(* IEC 61131-3 sources: AI4Industrial_Automation-FIRE2026/analysis/probe_reference, 30 files *)

(* ---- task_01.st ---- *)
PROGRAM T01
VAR_INPUT
    Low_Level_Sensor : BOOL;
    High_Level_Sensor : BOOL;
    Start_Button : BOOL;
    Stop_Button : BOOL;
END_VAR
VAR_OUTPUT
    Fill_Pump : BOOL;
END_VAR
Fill_Pump := ((Start_Button AND NOT Low_Level_Sensor) OR Fill_Pump) AND NOT High_Level_Sensor AND NOT Stop_Button;
END_PROGRAM

(* ---- task_02.st ---- *)
PROGRAM T02
VAR_OUTPUT
    Red_Light : BOOL;
    Yellow_Light : BOOL;
    Green_Light : BOOL;
END_VAR
VAR
    Cyc : TON;
    Restart : BOOL;
END_VAR
Cyc(IN := NOT Restart, PT := T#12s);
Restart := Cyc.Q;
Red_Light := Cyc.ET < T#5s;
Green_Light := Cyc.ET >= T#5s AND Cyc.ET < T#10s;
Yellow_Light := Cyc.ET >= T#10s;
END_PROGRAM

(* ---- task_03.st ---- *)
PROGRAM T03
VAR_INPUT
    Start_Button : BOOL;
    Stop_Button : BOOL;
    Overload_Trip : BOOL;
    Reset_Button : BOOL;
END_VAR
VAR_OUTPUT
    Motor_Run : BOOL;
    Fault_Lamp : BOOL;
END_VAR
IF Overload_Trip THEN
    Fault_Lamp := TRUE;
ELSIF Reset_Button THEN
    Fault_Lamp := FALSE;
END_IF;
Motor_Run := (Start_Button OR Motor_Run) AND NOT Stop_Button AND NOT Fault_Lamp;
END_PROGRAM

(* ---- task_04.st ---- *)
PROGRAM T04
VAR_INPUT
    Start_Button : BOOL;
    Stop_Button : BOOL;
    Bottle_Present : BOOL;
    Level_Sensor : BOOL;
END_VAR
VAR_OUTPUT
    Fill_Valve : BOOL;
    Bottle_Count : INT;
END_VAR
VAR
    Running : BOOL;
    Full_Edge : R_TRIG;
END_VAR
IF Start_Button THEN Running := TRUE; END_IF;
IF Stop_Button THEN Running := FALSE; Bottle_Count := 0; END_IF;
Fill_Valve := Running AND Bottle_Present AND NOT Level_Sensor;
Full_Edge(CLK := Running AND Bottle_Present AND Level_Sensor);
IF Full_Edge.Q THEN Bottle_Count := Bottle_Count + 1; END_IF;
END_PROGRAM

(* ---- task_05.st ---- *)
PROGRAM T05
VAR_INPUT
    Low_Level_Sensor : BOOL;
    High_Level_Sensor : BOOL;
    Auto_Mode : BOOL;
END_VAR
VAR_OUTPUT
    Auger_Motor : BOOL;
    High_Alarm : BOOL;
END_VAR
VAR
    T_High : TON;
END_VAR
Auger_Motor := Auto_Mode AND Low_Level_Sensor AND NOT High_Level_Sensor;
T_High(IN := High_Level_Sensor, PT := T#10s);
High_Alarm := T_High.Q;
END_PROGRAM

(* ---- task_06.st ---- *)
PROGRAM T06
VAR_INPUT
    Start_Button : BOOL;
    Stop_Button : BOOL;
    E_Stop : BOOL;
    Reset_Button : BOOL;
END_VAR
VAR_OUTPUT
    Motor_Run : BOOL;
    EStop_Lamp : BOOL;
END_VAR
IF E_Stop THEN
    EStop_Lamp := TRUE;
ELSIF Reset_Button THEN
    EStop_Lamp := FALSE;
END_IF;
Motor_Run := (Start_Button OR Motor_Run) AND NOT Stop_Button AND NOT EStop_Lamp;
END_PROGRAM

(* ---- task_07.st ---- *)
PROGRAM T07
VAR_INPUT
    Start_Button : BOOL;
    Stop_Button : BOOL;
    Speed_Select : BOOL;
    Low_Speed_Set : INT;
    High_Speed_Set : INT;
END_VAR
VAR_OUTPUT
    Conveyor_Speed : INT;
    Running_Lamp : BOOL;
END_VAR
VAR
    Running : BOOL;
END_VAR
Running := (Start_Button OR Running) AND NOT Stop_Button;
IF NOT Running THEN
    Conveyor_Speed := 0;
ELSIF Speed_Select THEN
    Conveyor_Speed := High_Speed_Set;
ELSE
    Conveyor_Speed := Low_Speed_Set;
END_IF;
Running_Lamp := Running;
END_PROGRAM

(* ---- task_08.st ---- *)
PROGRAM T08
VAR_INPUT
    Start_Button : BOOL;
    Reset_Button : BOOL;
    Level_A_Full : BOOL;
    Level_B_Full : BOOL;
END_VAR
VAR_OUTPUT
    Ingredient_A_Valve : BOOL;
    Ingredient_B_Valve : BOOL;
    Mixer_Motor : BOOL;
    Batch_Complete : BOOL;
END_VAR
VAR
    Filling : BOOL;
    Mixing : BOOL;
    T_Mix : TON;
END_VAR
IF Start_Button AND NOT Filling AND NOT Mixing AND NOT Batch_Complete THEN Filling := TRUE; END_IF;
Ingredient_A_Valve := Filling AND NOT Level_A_Full;
Ingredient_B_Valve := Filling AND NOT Level_B_Full;
IF Filling AND Level_A_Full AND Level_B_Full THEN Filling := FALSE; Mixing := TRUE; END_IF;
T_Mix(IN := Mixing, PT := T#30s);
IF T_Mix.Q THEN Mixing := FALSE; Batch_Complete := TRUE; END_IF;
Mixer_Motor := Mixing;
IF Reset_Button THEN Batch_Complete := FALSE; Filling := FALSE; Mixing := FALSE; END_IF;
END_PROGRAM

(* ---- task_09.st ---- *)
PROGRAM T09
VAR_INPUT
    Open_Button : BOOL;
    Close_Button : BOOL;
    Open_Limit : BOOL;
    Closed_Limit : BOOL;
    Obstacle_Sensor : BOOL;
END_VAR
VAR_OUTPUT
    Door_Motor_Open : BOOL;
    Door_Motor_Close : BOOL;
END_VAR
IF Door_Motor_Close AND Obstacle_Sensor THEN
    Door_Motor_Close := FALSE;
    Door_Motor_Open := TRUE;
END_IF;
IF Open_Button AND NOT Door_Motor_Close THEN Door_Motor_Open := TRUE; END_IF;
IF Close_Button AND NOT Door_Motor_Open THEN Door_Motor_Close := TRUE; END_IF;
IF Open_Limit THEN Door_Motor_Open := FALSE; END_IF;
IF Closed_Limit THEN Door_Motor_Close := FALSE; END_IF;
END_PROGRAM

(* ---- task_10.st ---- *)
PROGRAM T10
VAR_INPUT
    Car_Present : BOOL;
    Start_Button : BOOL;
END_VAR
VAR_OUTPUT
    Wash_Pump : BOOL;
    Rinse_Valve : BOOL;
    Dryer_Fan : BOOL;
    Cycle_Complete : BOOL;
END_VAR
VAR
    Step : INT;
    T_Step : TON;
END_VAR
CASE Step OF
    0:
        IF Car_Present AND Start_Button THEN Step := 1; END_IF;
    1:
        T_Step(IN := TRUE, PT := T#20s);
        IF T_Step.Q THEN T_Step(IN := FALSE); Step := 2; END_IF;
    2:
        T_Step(IN := TRUE, PT := T#15s);
        IF T_Step.Q THEN T_Step(IN := FALSE); Step := 3; END_IF;
    3:
        T_Step(IN := TRUE, PT := T#10s);
        IF T_Step.Q THEN T_Step(IN := FALSE); Step := 4; END_IF;
    4:
        IF NOT Car_Present THEN Step := 0; END_IF;
END_CASE;
Wash_Pump := Step = 1;
Rinse_Valve := Step = 2;
Dryer_Fan := Step = 3;
Cycle_Complete := Step = 4;
END_PROGRAM

(* ---- task_11.st ---- *)
PROGRAM T11
VAR_INPUT
    Box_Sensor : BOOL;
END_VAR
VAR_OUTPUT
    Pusher_Cylinder : BOOL;
    Box_Count_Display : INT;
END_VAR
VAR
    Cnt : CTU;
    Push : TP;
END_VAR
Cnt(CU := Box_Sensor, R := Cnt.Q, PV := 5);
Push(IN := Cnt.Q, PT := T#1s);
Cnt(CU := Box_Sensor, R := Cnt.Q, PV := 5);
Pusher_Cylinder := Push.Q;
Box_Count_Display := Cnt.CV;
END_PROGRAM

(* ---- task_12.st ---- *)
PROGRAM T12
VAR_INPUT
    Weight_Input : INT;
    Target_Weight : INT;
    Photo_Eye : BOOL;
END_VAR
VAR_OUTPUT
    Reject_Pusher : BOOL;
END_VAR
VAR
    Trig : R_TRIG;
    Pulse : TP;
END_VAR
Trig(CLK := Photo_Eye);
Pulse(IN := Trig.Q AND ABS(Weight_Input - Target_Weight) > 5, PT := T#500ms);
Reject_Pusher := Pulse.Q;
END_PROGRAM

(* ---- task_13.st ---- *)
PROGRAM T13
VAR_INPUT
    Temp_Sensor : INT;
    Setpoint : INT;
END_VAR
VAR_OUTPUT
    Heater : BOOL;
END_VAR
IF Temp_Sensor < Setpoint - 5 THEN Heater := TRUE;
ELSIF Temp_Sensor > Setpoint + 5 THEN Heater := FALSE; END_IF;
END_PROGRAM

(* ---- task_14.st ---- *)
PROGRAM T14
VAR_INPUT
    Temp_Sensor : INT;
END_VAR
VAR_OUTPUT
    Fan1 : BOOL;
    Fan2 : BOOL;
END_VAR
IF Temp_Sensor > 300 THEN Fan1 := TRUE; ELSIF Temp_Sensor < 280 THEN Fan1 := FALSE; END_IF;
IF Temp_Sensor > 350 THEN Fan2 := TRUE; ELSIF Temp_Sensor < 330 THEN Fan2 := FALSE; END_IF;
END_PROGRAM

(* ---- task_15.st ---- *)
PROGRAM T15
VAR_INPUT
    Pressure_Sensor : INT;
END_VAR
VAR_OUTPUT
    Compressor_Motor : BOOL;
END_VAR
IF Pressure_Sensor < 80 THEN Compressor_Motor := TRUE;
ELSIF Pressure_Sensor > 120 THEN Compressor_Motor := FALSE; END_IF;
END_PROGRAM

(* ---- task_16.st ---- *)
PROGRAM T16
VAR_INPUT
    CO2_Sensor : INT;
END_VAR
VAR_OUTPUT
    Damper_Position : INT;
END_VAR
IF CO2_Sensor <= 600 THEN Damper_Position := 0;
ELSIF CO2_Sensor >= 1000 THEN Damper_Position := 100;
ELSE Damper_Position := (CO2_Sensor - 600) * 100 / 400; END_IF;
END_PROGRAM

(* ---- task_17.st ---- *)
PROGRAM T17
VAR_INPUT
    Soil_Moisture : INT;
    Manual_Start : BOOL;
END_VAR
VAR_OUTPUT
    Irrigation_Valve : BOOL;
END_VAR
VAR
    Hold : TP;
END_VAR
Hold(IN := Soil_Moisture < 30 OR Manual_Start, PT := T#10m);
Irrigation_Valve := Hold.Q;
END_PROGRAM

(* ---- task_18.st ---- *)
PROGRAM T18
VAR_INPUT
    Part_Detect : BOOL;
    Part_Good : BOOL;
END_VAR
VAR_OUTPUT
    Reject_Cylinder : BOOL;
END_VAR
VAR
    Trig : R_TRIG;
    Pulse : TP;
END_VAR
Trig(CLK := Part_Detect);
Pulse(IN := Trig.Q AND NOT Part_Good, PT := T#500ms);
Reject_Cylinder := Pulse.Q;
END_PROGRAM

(* ---- task_19.st ---- *)
PROGRAM T19
VAR_INPUT
    Call_Floor1 : BOOL;
    Call_Floor2 : BOOL;
    At_Floor1 : BOOL;
    At_Floor2 : BOOL;
END_VAR
VAR_OUTPUT
    Motor_Up : BOOL;
    Motor_Down : BOOL;
END_VAR
Motor_Up := ((Call_Floor2 AND NOT At_Floor2) OR Motor_Up) AND NOT At_Floor2 AND NOT Motor_Down;
Motor_Down := ((Call_Floor1 AND NOT At_Floor1) OR Motor_Down) AND NOT At_Floor1 AND NOT Motor_Up;
END_PROGRAM

(* ---- task_20.st ---- *)
PROGRAM T20
VAR_INPUT
    Start_Cycle : BOOL;
    Part_Present : BOOL;
    Gripper_Extended : BOOL;
    Gripper_Retracted : BOOL;
END_VAR
VAR_OUTPUT
    Cylinder_Extend : BOOL;
    Gripper_Close : BOOL;
END_VAR
VAR
    Step : INT;
    Dwell : TON;
END_VAR
CASE Step OF
    0:
        IF Start_Cycle AND Part_Present THEN Step := 1; END_IF;
    1:
        IF Gripper_Extended THEN Step := 2; END_IF;
    2:
        Dwell(IN := TRUE, PT := T#500ms);
        IF Dwell.Q THEN Dwell(IN := FALSE); Step := 3; END_IF;
    3:
        IF Gripper_Retracted THEN Step := 0; END_IF;
END_CASE;
Cylinder_Extend := Step = 1 OR Step = 2;
Gripper_Close := Step = 2 OR Step = 3;
IF Step = 3 AND Gripper_Retracted THEN Gripper_Close := FALSE; END_IF;
IF Step = 0 THEN Gripper_Close := FALSE; END_IF;
END_PROGRAM

(* ---- task_21.st ---- *)
PROGRAM T21
VAR_INPUT
    Start_Button : BOOL;
    Stop_Button : BOOL;
    Light_Curtain_Clear : BOOL;
END_VAR
VAR_OUTPUT
    Conveyor_Run : BOOL;
    Safety_Fault_Lamp : BOOL;
END_VAR
Conveyor_Run := (Start_Button OR Conveyor_Run) AND NOT Stop_Button AND Light_Curtain_Clear;
Safety_Fault_Lamp := NOT Light_Curtain_Clear;
END_PROGRAM

(* ---- task_22.st ---- *)
PROGRAM T22
VAR_INPUT
    Start_Button : BOOL;
    Stop_Button : BOOL;
    Entry_Photo_Eye : BOOL;
    Exit_Photo_Eye : BOOL;
END_VAR
VAR_OUTPUT
    Conveyor_Run : BOOL;
    Jam_Alarm : BOOL;
END_VAR
VAR
    T_Jam : TON;
END_VAR
T_Jam(IN := Entry_Photo_Eye AND NOT Exit_Photo_Eye, PT := T#8s);
IF T_Jam.Q THEN Jam_Alarm := TRUE; END_IF;
IF Stop_Button THEN Jam_Alarm := FALSE; END_IF;
Conveyor_Run := (Start_Button OR Conveyor_Run) AND NOT Stop_Button AND NOT Jam_Alarm;
END_PROGRAM

(* ---- task_23.st ---- *)
PROGRAM T23
VAR_INPUT
    Start_Button : BOOL;
    Stop_Button : BOOL;
    Flow_A_Pulse : BOOL;
END_VAR
VAR_OUTPUT
    Valve_A : BOOL;
    Valve_B : BOOL;
END_VAR
VAR
    Running : BOOL;
    Cnt : CTU;
END_VAR
Running := (Start_Button OR Running) AND NOT Stop_Button;
Valve_A := Running;
Cnt(CU := Flow_A_Pulse AND Running, R := Cnt.Q AND NOT Flow_A_Pulse, PV := 4);
Valve_B := Running AND Cnt.Q;
END_PROGRAM

(* ---- task_24.st ---- *)
PROGRAM T24
VAR_INPUT
    Start_Button : BOOL;
    Stop_Button : BOOL;
END_VAR
VAR_OUTPUT
    Lamp1 : BOOL;
    Lamp2 : BOOL;
    Lamp3 : BOOL;
    Lamp4 : BOOL;
END_VAR
VAR
    Running : BOOL;
    Cyc : TON;
    Restart : BOOL;
END_VAR
Running := (Start_Button OR Running) AND NOT Stop_Button;
Cyc(IN := Running AND NOT Restart, PT := T#2s);
Restart := Cyc.Q;
Lamp1 := Running AND Cyc.ET < T#500ms;
Lamp2 := Running AND Cyc.ET >= T#500ms AND Cyc.ET < T#1s;
Lamp3 := Running AND Cyc.ET >= T#1s AND Cyc.ET < T#1500ms;
Lamp4 := Running AND Cyc.ET >= T#1500ms;
END_PROGRAM

(* ---- task_25.st ---- *)
PROGRAM T25
VAR_INPUT
    pH_Sensor : INT;
END_VAR
VAR_OUTPUT
    Acid_Pump : BOOL;
    Base_Pump : BOOL;
END_VAR
Acid_Pump := pH_Sensor > 720;
Base_Pump := pH_Sensor < 680;
END_PROGRAM

(* ---- task_26.st ---- *)
PROGRAM T26
VAR_INPUT
    Start_Button : BOOL;
    Stop_Button : BOOL;
END_VAR
VAR_OUTPUT
    Conveyor_Run : BOOL;
END_VAR
Conveyor_Run := (Start_Button OR Conveyor_Run) AND NOT Stop_Button;
END_PROGRAM

(* ---- task_27.st ---- *)
PROGRAM T27
VAR_INPUT
    RPM_Set : INT;
    Start_Button : BOOL;
    Stop_Button : BOOL;
END_VAR
VAR_OUTPUT
    Conveyor_Run : INT;
    start_light : BOOL;
END_VAR
start_light := (Start_Button OR start_light) AND NOT Stop_Button;
IF start_light THEN Conveyor_Run := RPM_Set; ELSE Conveyor_Run := 0; END_IF;
END_PROGRAM

(* ---- task_28.st ---- *)
PROGRAM T28
VAR_INPUT
    RPM_Set : INT;
    Start_Button : BOOL;
    Stop_Button : BOOL;
END_VAR
VAR_OUTPUT
    Digital_Display : INT;
    Conveyor_Run : INT;
END_VAR
VAR
    Running : BOOL;
END_VAR
Running := (Start_Button OR Running) AND NOT Stop_Button;
IF Running THEN Conveyor_Run := RPM_Set; ELSE Conveyor_Run := 0; END_IF;
Digital_Display := RPM_Set;
END_PROGRAM

(* ---- task_29.st ---- *)
PROGRAM T29
VAR_INPUT
    RPM_Set : INT;
    Start_Button : BOOL;
    Stop_Button : BOOL;
    Vision_Sensor : INT;
END_VAR
VAR_OUTPUT
    Conveyor_Run : INT;
    start_light : BOOL;
    Digital_Display : INT;
    display_box_counter : INT;
END_VAR
start_light := (Start_Button OR start_light) AND NOT Stop_Button;
IF start_light THEN Conveyor_Run := RPM_Set; ELSE Conveyor_Run := 0; END_IF;
Digital_Display := RPM_Set;
END_PROGRAM

(* ---- task_30.st ---- *)
PROGRAM T30
VAR_INPUT
    RPM_Set : INT;
    Start_Button : BOOL;
    Stop_Button : BOOL;
    Vision_Sensor : INT;
END_VAR
VAR_OUTPUT
    Conveyor_Run : INT;
    start_light : BOOL;
    Digital_Display : INT;
    display_box_counter : INT;
    blue_box_counter : INT;
    grey_box_counter : INT;
    green_box_counter : INT;
END_VAR
start_light := (Start_Button OR start_light) AND NOT Stop_Button;
IF start_light THEN Conveyor_Run := RPM_Set; ELSE Conveyor_Run := 0; END_IF;
Digital_Display := RPM_Set;
END_PROGRAM
